(*
    This testsuite tests the different assert-functions for all the different data types in TwinCAT.
    For every data type at least two different tests have been defined:
        1. One test that succeeds (Expected and actual are equal)
        2. One test that fails (Expected and actual are false).
*)
{attribute 'call_after_init'}
FUNCTION_BLOCK FB_NewTestFB_Test EXTENDS TcUnit.FB_TestSuite IMPLEMENTS TcUnit.I_RunnableTestSuite
VAR
    Assert : TcUnit.FB_Assert;
    
    testTestSuite: UnitTestSuite;
    testFB: UnitTest(testTestSuite);
END_VAR

METHOD FB_init : BOOL
VAR_INPUT
	bInitRetains : BOOL; // if TRUE, the retain variables are initialized (warm start / cold start)
	bInCopyCode : BOOL;  // if TRUE, the instance afterwards gets moved into the copy code (online change)
END_VAR
SUPER^.RegisterTestSuite(THIS^);
END_METHOD

METHOD RunTests : TCUNIT.E_TestSuiteRunState
Test_GetTestSuiteUninitialized();
Test_GetTestSuiteInitialized();

RunTests := TCUNIT.E_TestSuiteRunState.FINISHED;
END_METHOD

METHOD Test_GetTestSuiteInitialized
VAR
    expected: UDINT;
    actual: UDINT;
END_VAR
VAR_INST
    testIntf: ITestSuite;
END_VAR
TEST('Test_GetTestSuiteInitialized');

expected := TO_UDINT(ADR(testTestSuite));
testIntf := testFB.testSuite;
actual := TO_UDINT(ADR(testIntf));

Assert.AssertEquals_UDINT(expected, actual, 'Initialized UnitTest is wrong');
END_METHOD

METHOD Test_GetTestSuiteUninitialized
VAR
    expected: UDINT;
    actual: UDINT;
END_VAR
VAR_INST
    testFB: UnitTest(0);
    testIntf: ITestSuite;
END_VAR
TEST('Test_GetTestSuiteUninitialized');

expected := 0;
testIntf := testFB.testSuite;
actual := TO_UDINT(ADR(testIntf));

Assert.AssertEquals_UDINT(expected, actual, 'Uninitialized UnitTest is non zero');
END_METHOD

END_FUNCTION_BLOCK

(* stored: Version 1.1.0.1, ProductVersion 3.1.4022.12
   POU FB_NewTestFB_Test: Id {e26b3756-9357-4d27-8f4d-66820ebee40b}, SpecialFunc None
   Method FB_init: Id {fb3fd669-9f91-48e1-811f-7e7a9a1556f5}
   Method RunTests: Id {f3839f6c-e99d-404b-b0db-30f053091682}
   Method Test_GetTestSuiteInitialized: Id {e35cf077-d735-4287-b16e-2b0973a1c88f}
   Method Test_GetTestSuiteUninitialized: Id {d1b86bd3-130d-4c25-a228-4a0507fa9288} *)
